ABB RAPID module: sbt_comm003.mod

module sbt_comm003
!***********************************************************
!
! Copyright 2018 - 2024 speedbot All Rights reserved.
!
! file Name: sbt_comm003
!
!  Description:
!    Language             ==   Rapid for ABB ROBOT
!    Date                 ==   2024 - 06 - 17
!    Modification Data    ==   2024 - 06 - 17
!
!  Author: speedbot
!
!  Version: 3.0
! ***********************************************************

local var busin_t BusInput := [0, 0, 0, 0, 0, 0, 0, 0, 0, 0, 0, 0, 0, 0, 0];
local var busout_t BusOutput := [0, 0, 0, 0, 0, 0, 0, 0, 0, 0, 0, 0, 0, 0, 0];

local var num BusTimeout := 5;

local var cmd_typ03_t CmdType03 := [0,0,0,0,0,0,0,0,0,0,0,0,0,0,0,0,0,0];
local var cmd_typ01_t CmdType01 := [0, 0, 0, 0, 0, 0, 0.0, 0.0];

local var errnum Res := 0;

pers byte VinComm003{17};

proc sbt_comm003_(\switch CMD_VPARAM | switch CMD_POS | switch CMD_TRIG | switch CMD_SCANSRT | switch CMD_SCANSTP |switch CMD_END,
                  \byte Pid, \byte Vin{*},
                  \byte PictureId,
                  \inout robtarget ThisPos)

    var errnum Res := -1;

    while true do

        ! waittime \InPos, 0.0;

        if present(CMD_VPARAM) then

            log_clear_;

            bus_init_ BusInput, BusOutput, \RobId := 0, \ProtId := PTC_GEN_CMD;

            CmdType03 := [0,0,0,0,0,0,0,0,0,0,0,0,0,0,0,0,0,0];

            CmdType01 := [0, 0, 0, 0, 0, 0, 0.0, 0.0];

            if present(Pid) then
                CmdType03.byte01 := Pid;
            endif

            if present(Vin) then

                CmdType03.byte02 := Vin{1};
                CmdType03.byte03 := Vin{2};
                CmdType03.byte04 := Vin{3};
                CmdType03.byte05 := Vin{4};
                CmdType03.byte06 := Vin{5};
                CmdType03.byte07 := Vin{6};
                CmdType03.byte08 := Vin{7};
                CmdType03.byte09 := Vin{8};
                CmdType03.byte10 := Vin{9};
                CmdType03.byte11 := Vin{10};
                CmdType03.byte12 := Vin{11};
                CmdType03.byte13 := Vin{12};
                CmdType03.byte14 := Vin{13};
                CmdType03.byte15 := Vin{14};
                CmdType03.byte16 := Vin{15};
                CmdType03.byte17 := Vin{16};
                CmdType03.byte18 := Vin{17};
            endif

            Res := bus_cmd137_(BUSCMD_WRITE, BUSCMD_MST, BusInput, BusOutput, CmdType03);
            Res := bus_cmd001_(BUSCMD_READ, BUSCMD_MST, BusInput, BusOutput, \Timeout := BusTimeout);

            if Res = 0 then

                return;
            else

                err_display_ BusInput,BusOutput;
            endif
        endif

        if present(CMD_TRIG) or present(CMD_SCANSRT) or present(CMD_SCANSTP) then

            waittime \InPos, 0.0;

            if present(CMD_TRIG) then
                CmdType01.Byte01 := 1;
            endif

            if present(CMD_SCANSRT) then
                CmdType01.Byte01 := 2;
            endif

            if present(CMD_SCANSTP) then
                CmdType01.Byte01 := 3;
            endif

            CmdType01.Byte02 := 0;
            if present(PictureId) then
                CmdType01.Short03 := PictureId;
            else
                CmdType01.Short03 := 0;
            endif
            CmdType01.Short04 := 0;
            CmdType01.Int05 := 0;
            CmdType01.Int06 := 0;
            CmdType01.Float07 := 0;
            CmdType01.Float08 := 0;

            Res := bus_cmd012_(BUSCMD_WRITE, BUSCMD_MST, BusInput, BusOutput, CmdType01);
            Res := bus_cmd001_(BUSCMD_READ, BUSCMD_MST, BusInput, BusOutput, \Timeout := BusTimeout);

            if Res = 0 then

            else
                err_display_ BusInput,BusOutput;
            endif
            return;
        endif

        if present(CMD_POS) then

            CmdType01 := [0, 0, 0, 0, 0, 0, 0.0, 0.0];

            Res := bus_cmd021_(BUSCMD_WRITE, BUSCMD_MST, BusInput, BusOutput, CmdType01);
            Res := bus_cmd129_(BUSCMD_READ, BUSCMD_MST, BusInput, BusOutput, ThisPos, \Timeout := BusTimeout);

            if Res = 0 then

                 return;
            else

                err_display_ BusInput,BusOutput;
                bus_init_ BusInput, BusOutput, \RobId := 0, \ProtId := PTC_GEN_CMD;
            endif

        endif

        if present(CMD_END) then

            CmdType01 := [100, 0, 0, 0, 0, 0, 0.0, 0.0];

            Res := bus_cmd013_(BUSCMD_WRITE, BUSCMD_MST, BusInput, BusOutput, CmdType01);
            Res := bus_cmd001_(BUSCMD_READ, BUSCMD_MST, BusInput, BusOutput, \Timeout := BusTimeout);

            if Res = 0 then

            else

                err_display_ BusInput,BusOutput;
            endif

            return;
        endif

        log_error_ \Tag := "999", "Calibration Param Err", \ELOG;
    endwhile

endproc

local proc err_display_(busin_t BusIn,busout_t BusOut)

    if  BusIn.SysReady = 0 then

        log_error_ \Tag := "901", "Software not ready", \ELOG;
        return;
    endif

    if BusIn.TellId <> BusOut.RobTellId then

        log_error_ \Tag := "902", "Software processing timeout", \ELOG;
    endif

    test BusIn.ErrorId

    case 1:
        log_error_ \Tag := "001", "Camera connection failed", \ELOG;
    case 2:
        log_warn_ \Tag := "002", "Camera shot failed", \ELOG;
    case 3:
        log_error_ \Tag := "003", "Error correction failure", \ELOG;
    case 4:
        log_warn_ \Tag := "004", "Gap surface difference failed", \ELOG;
    default :
        log_error_ \Tag := "903", "Unknow error", \ELOG;
    endtest

endproc

endmodule
